TYPE ST_ConfigurableCylinderParCmd :
STRUCT
    Reserved : BOOL;
END_STRUCT
END_TYPE

(* stored: Version 1.1.0.1, ProductVersion 3.1.4024.12
   DUT ST_ConfigurableCylinderParCmd: Id {087542c5-d88f-4772-9591-aecbe090436b} *)
